// Mitsubishi GX Works2 project: wor01052023   PLC: FX3G

// global labels: Global1
VAR_GLOBAL
  X_3 AT X003 : BOOL;
  Temp_Under15 AT X002 : BOOL;
  Machine_On AT Y004 : BOOL;
  Force_Stop AT X005 : BOOL;
  Cream_Storage AT D1145 : INT;
  M_19 AT M19 : BOOL;
  M_18 AT M18 : BOOL;
END_VAR
VAR_GLOBAL CONSTANT
  biscuits_6 : INT := 6;
END_VAR
VAR_GLOBAL
  biscuits_storage AT D1150 : INT;
  Camera_sensor AT X004 : BOOL;
  Touch_sensor AT X001 : BOOL;
  M_20 AT M20 : BOOL;
  Move_cream AT X011 : BOOL;
  Y_1 AT Y001 : BOOL;
  M_8 AT M8 : BOOL;
END_VAR
VAR_GLOBAL CONSTANT
  RE_timer1 : INT := 10;
END_VAR
VAR_GLOBAL
  TC4_lights AT TC4 : BOOL;
  Y_0 AT Y000 : BOOL;
  TC5_lights AT TC5 : BOOL;
  TS5 AT TS5 : BOOL;
  TC1_lights AT TC1 : BOOL;
  TS1 AT TS1 : BOOL;
END_VAR
VAR_GLOBAL CONSTANT
  RE_timer2 : INT := 40;
END_VAR
VAR_GLOBAL
  M_9 AT M9 : BOOL;
  TS4 AT TS4 : BOOL;
  Chocolate_Container AT D1138 : INT;
  Icing_container AT D1120 : INT;
  Input_chocolate AT D2000 : INT;
  Input_icing AT D2100 : INT;
  Input_biscuits AT D2200 : INT;
  M_88 AT M88 : BOOL;
  Min_chocolate AT D2300 : INT;
  Min_Icing AT D2400 : INT;
  Min_biscuits AT D2500 : INT;
END_VAR
VAR_GLOBAL CONSTANT
  Cream_300 : INT := 300;
END_VAR
VAR_GLOBAL
  M_89 AT M89 : BOOL;
  M_90 AT M90 : BOOL;
  M_91 AT M91 : BOOL;
  CC_0 AT CC0 : BOOL;
  CC_1 AT CC1 : BOOL;
  M_111 AT M111 : BOOL;
  M_112 AT M112 : BOOL;
END_VAR
VAR_GLOBAL CONSTANT
  Double_Cover240 : INT := 240;
  Min_1 : INT := 1;
END_VAR
VAR_GLOBAL
  Y_7 AT Y007 : BOOL;
  Start_day AT X007 : BOOL;
  M_404 AT M404 : BOOL;
  X_10 AT X010 : BOOL;
  X_0 AT X000 : BOOL;
  Counter_5 AT CC5 : BOOL;
END_VAR
VAR_GLOBAL CONSTANT
  RE_counter : INT := 5;
END_VAR
VAR_GLOBAL
  CS5_counter AT CS5 : BOOL;
  Y_2 AT Y002 : BOOL;
  Counter_1 AT CC1 : BOOL;
END_VAR
VAR_GLOBAL CONSTANT
  RE_counter1 : INT := 1;
END_VAR
VAR_GLOBAL
  Counter_6 AT CC6 : BOOL;
END_VAR
VAR_GLOBAL CONSTANT
  RE_count6 : INT := 6;
END_VAR
VAR_GLOBAL
  CS6_downCounter AT CS6 : BOOL;
  finish_packing AT M16 : BOOL;  (* after packing 6 creamBos we will send a signal to add them to the total *)
  analog_output AT D8282 : INT;
  M_17 AT M17 : BOOL;  (* after packing 6 creamBos we will send a signal to add them to the total *)
END_VAR
VAR_GLOBAL CONSTANT
  CreamBo_Unit : INT := 6;
END_VAR
VAR_GLOBAL
  Y_3 AT Y003 : BOOL;
  global_num_CreamBos AT D1234 : INT;
END_VAR
VAR_GLOBAL CONSTANT
  Const_10 : INT := 10;
END_VAR
VAR_GLOBAL
  end_of_day AT M200 : BOOL;
  M_301 AT M301 : BOOL;
  TC11_lights AT TC11 : BOOL;
END_VAR
VAR_GLOBAL CONSTANT
  RE_timer11 : INT := 40;
END_VAR
VAR_GLOBAL
  TS11 AT TS11 : BOOL;
  M_500 AT M500 : BOOL;
  M_501 AT M501 : BOOL;
  TS12 AT TS12 : BOOL;
  TC12_lights AT TC12 : BOOL;
END_VAR
VAR_GLOBAL CONSTANT
  RE_timer12 : INT := 10;
END_VAR
VAR_GLOBAL
  TS13 AT TS13 : BOOL;
  M_505 AT M505 : BOOL;
  TC13_lights AT TC13 : BOOL;
END_VAR
VAR_GLOBAL CONSTANT
  RE_timer13 : INT := 10;
END_VAR
VAR_GLOBAL
  X_6 AT X006 : BOOL;
  Analog_Input AT D8280 : INT;
  TC_DipTimer AT TC20 : BOOL;
END_VAR
VAR_GLOBAL CONSTANT
  RE_5secTimer : INT := 50;  (* 50 mili seconds is 5 seconds *)
END_VAR
VAR_GLOBAL
  TS1_timer AT TS20 : BOOL;
END_VAR
VAR_GLOBAL CONSTANT
  constant6 : INT := 6;
  constant5 : INT := 5;
END_VAR
VAR_GLOBAL
  Container_Dip AT D1139 : INT;
END_VAR
VAR_GLOBAL CONSTANT
  Regular_Cover120 : INT := 120;
END_VAR
VAR_GLOBAL
  M_101 AT M101 : BOOL;
  Y_4 AT Y004 : BOOL;
  M_120 AT M120 : BOOL;
  M_99 AT M99 : BOOL;
  M_113 AT M113 : BOOL;
  M_102 AT M102 : BOOL;
  CS_0 AT CS0 : BOOL;
  CS_1 AT CS1 : BOOL;
  M_300 AT M300 : BOOL;
END_VAR
VAR_GLOBAL CONSTANT
  constant_390 : INT := 390;
END_VAR
VAR_GLOBAL
  Input_moveNew AT D2270 : INT;
  M_75 AT M75 : BOOL;
  TS20_timer AT TS20 : BOOL;
  M_405 AT M405 : BOOL;
  M_321 AT M321 : BOOL;
  M_322 AT M322 : BOOL;
  M_323 AT M323 : BOOL;
  M_324 AT M324 : BOOL;
  M_325 AT M325 : BOOL;
  output_test AT D1237 : INT;
  output_mul AT D1238 : INT;
  M_80 AT M80 : BOOL;
  M_333 AT M333 : BOOL;
END_VAR

// task Task_01 (event TRUE, interval 0, priority 31): POU_01

PROGRAM POU_01
VAR
  M_0 : BOOL;
  TS2 : BOOL;
END_VAR
(* structured ladder/FBD written out as ST: instructions are called as NAME(EN, inputs, outputs); _pN, _eN, _tN stand for wires *)
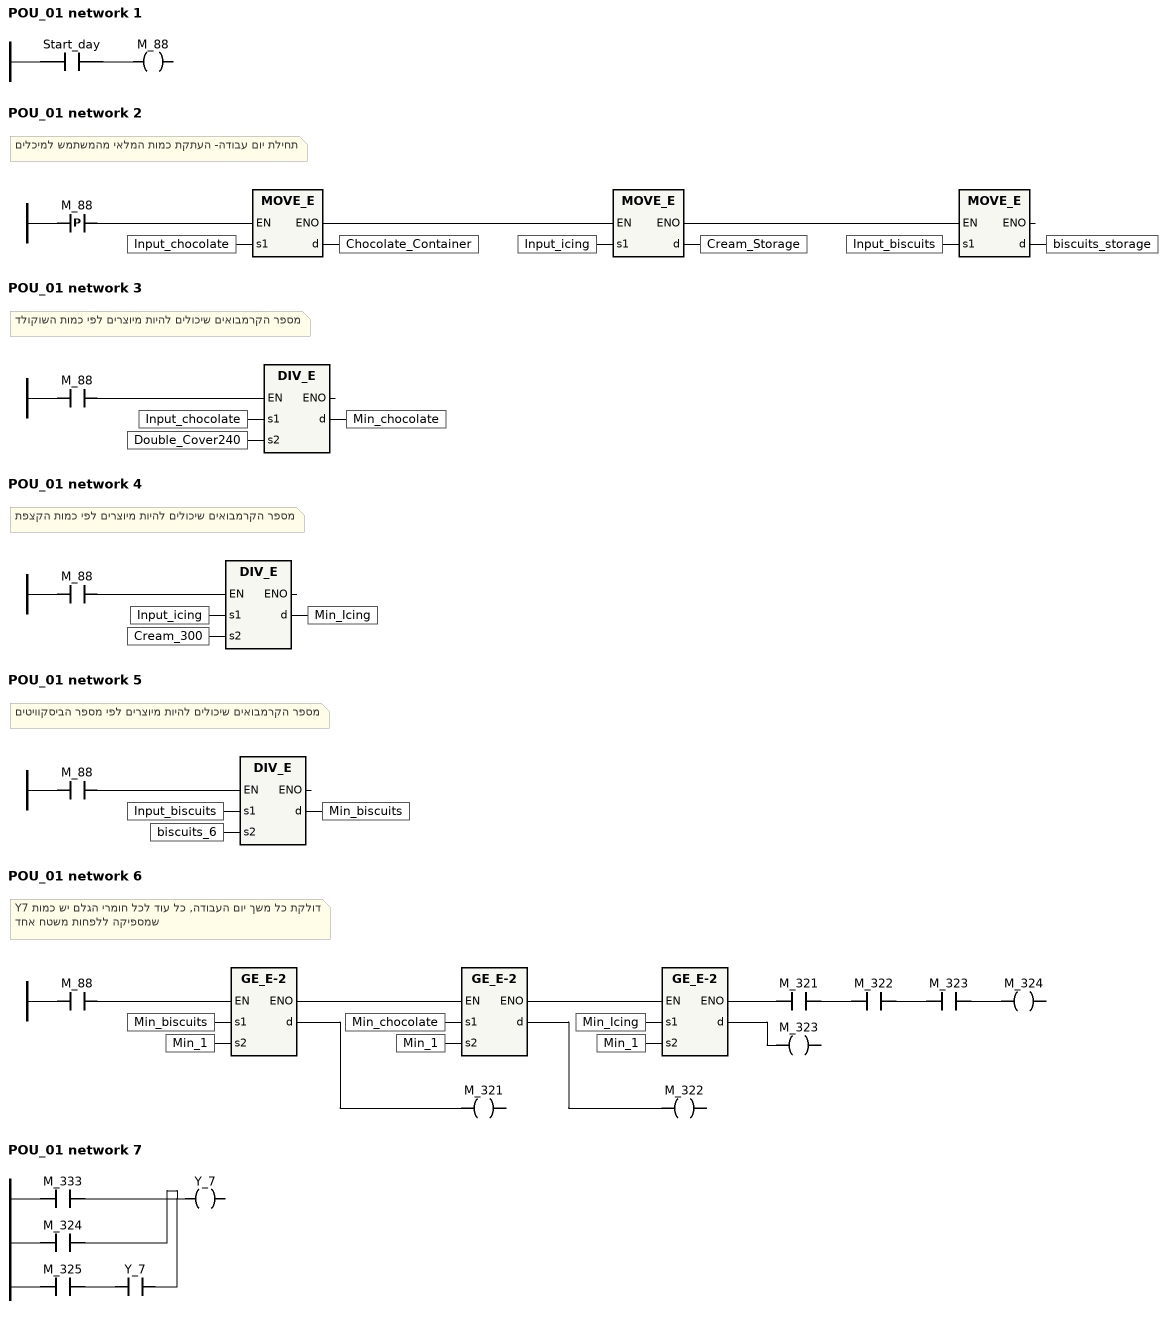
(* network 1 *)
M_88 := Start_day;
(* network 2 *)
(* תחילת יום עבודה- העתקת כמות המלאי מהמשתמש למיכלים *)
_e1 := MOVE_E(LDP(TRUE, M_88), Input_chocolate, Chocolate_Container);
_e2 := MOVE_E(_e1, Input_icing, Cream_Storage);
MOVE_E(_e2, Input_biscuits, biscuits_storage);
(* network 3 *)
(* מספר הקרמבואים שיכולים להיות מיוצרים לפי כמות השוקולד *)
DIV_E(M_88, Input_chocolate, Double_Cover240, Min_chocolate);
(* network 4 *)
(* מספר הקרמבואים שיכולים להיות מיוצרים לפי כמות הקצפת *)
DIV_E(M_88, Input_icing, Cream_300, Min_Icing);
(* network 5 *)
(* מספר הקרמבואים שיכולים להיות מיוצרים לפי מספר הביסקוויטים *)
DIV_E(M_88, Input_biscuits, biscuits_6, Min_biscuits);
(* network 6 *)
(* Y7 דולקת כל משך יום העבודה, כל עוד לכל חומרי הגלם יש כמות שמספיקה ללפחות משטח אחד *)
_e2 := GE_E(M_88, Min_biscuits, Min_1, _t1);
_e4 := GE_E(_e2, Min_chocolate, Min_1, _t3);
_e6 := GE_E(_e4, Min_Icing, Min_1, _t5);
M_324 := _e6 AND M_321 AND M_322 AND M_323;
M_321 := _t1;
M_323 := _t5;
M_322 := _t3;
(* network 7 *)
Y_7 := M_333 OR M_324 OR (M_325 AND Y_7);
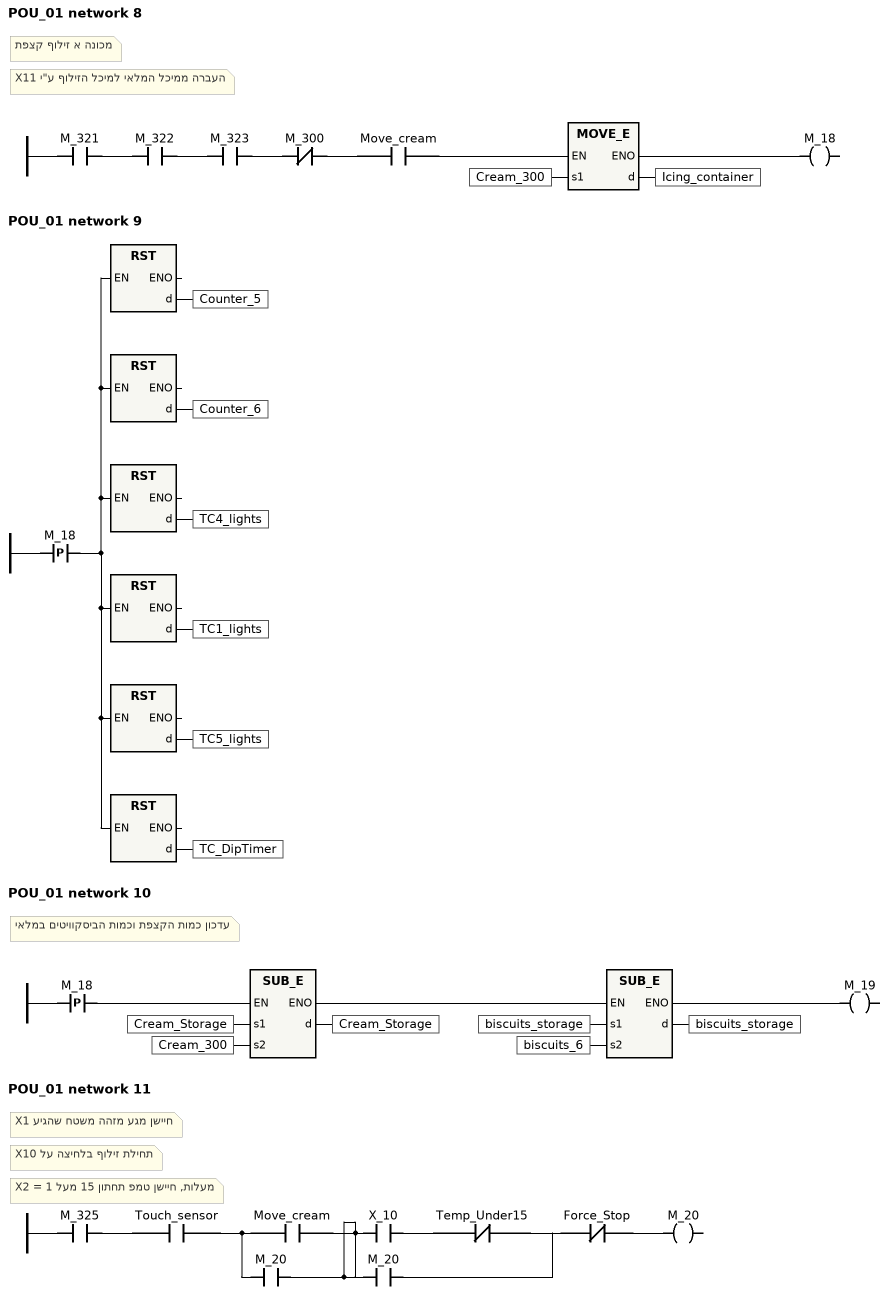
(* network 8 *)
(* מכונה א זילוף קצפת *)
(* העברה ממיכל המלאי למיכל הזילוף ע"י X11 *)
_e1 := MOVE_E(M_321 AND M_322 AND M_323 AND NOT M_300 AND Move_cream, Cream_300, Icing_container);
M_18 := _e1;
(* network 9 *)
_p1 := LDP(TRUE, M_18);
RST(_p1, Counter_5);
RST(_p1, Counter_6);
RST(_p1, TC4_lights);
RST(_p1, TC1_lights);
RST(_p1, TC5_lights);
RST(_p1, TC_DipTimer);
(* network 10 *)
(* עדכון כמות הקצפת וכמות הביסקוויטים במלאי *)
_e1 := SUB_E(LDP(TRUE, M_18), Cream_Storage, Cream_300, Cream_Storage);
_e2 := SUB_E(_e1, biscuits_storage, biscuits_6, biscuits_storage);
M_19 := _e2;
(* network 11 *)
(* חיישן מגע מזהה משטח שהגיע X1 *)
(* תחילת זילוף בלחיצה על X10 *)
(* X2 = 1 מעל 15 מעלות, חיישן טמפ תחתון *)
_p1 := M_325 AND Touch_sensor;
_p2 := (_p1 AND Move_cream) OR (_p1 AND M_20);
M_20 := ((_p2 AND X_10 AND NOT Temp_Under15) OR (_p2 AND M_20)) AND NOT Force_Stop;
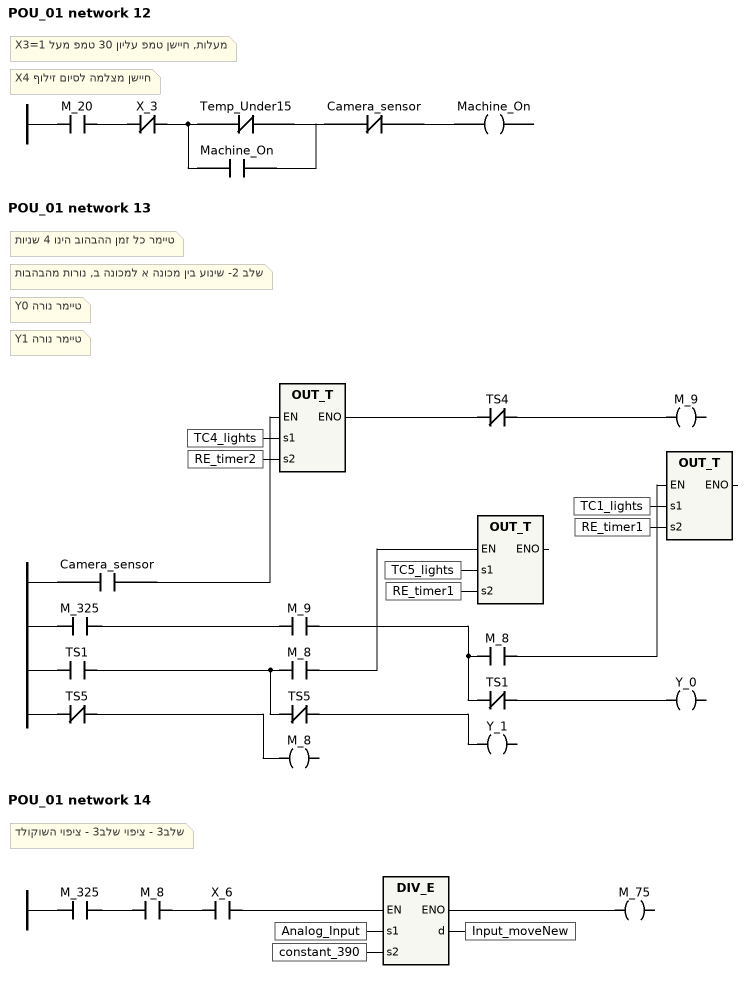
(* network 12 *)
(* X3=1 טמפ מעל 30 מעלות, חיישן טמפ עליון *)
(* חיישן מצלמה לסיום זילוף X4 *)
_p1 := M_20 AND NOT X_3;
Machine_On := ((_p1 AND NOT Temp_Under15) OR (_p1 AND Machine_On)) AND NOT Camera_sensor;
(* network 13 *)
(* טיימר כל זמן ההבהוב הינו 4 שניות *)
(* שלב 2- שינוע בין מכונה א למכונה ב, נורות מהבהבות *)
(* טיימר נורה Y0 *)
(* טיימר נורה Y1 *)
_e1 := OUT_T(Camera_sensor, TC4_lights, RE_timer2);
M_9 := _e1 AND NOT TS4;
_p2 := M_325 AND M_9;
OUT_T(_p2 AND M_8, TC1_lights, RE_timer1);
Y_0 := _p2 AND NOT TS1;
OUT_T(TS1 AND M_8, TC5_lights, RE_timer1);
Y_1 := TS1 AND NOT TS5;
M_8 := NOT TS5;
(* network 14 *)
(* שלב3 - ציפוי שלב3 - ציפוי השוקולד *)
_e1 := DIV_E(M_325 AND M_8 AND X_6, Analog_Input, constant_390, Input_moveNew);
M_75 := _e1;
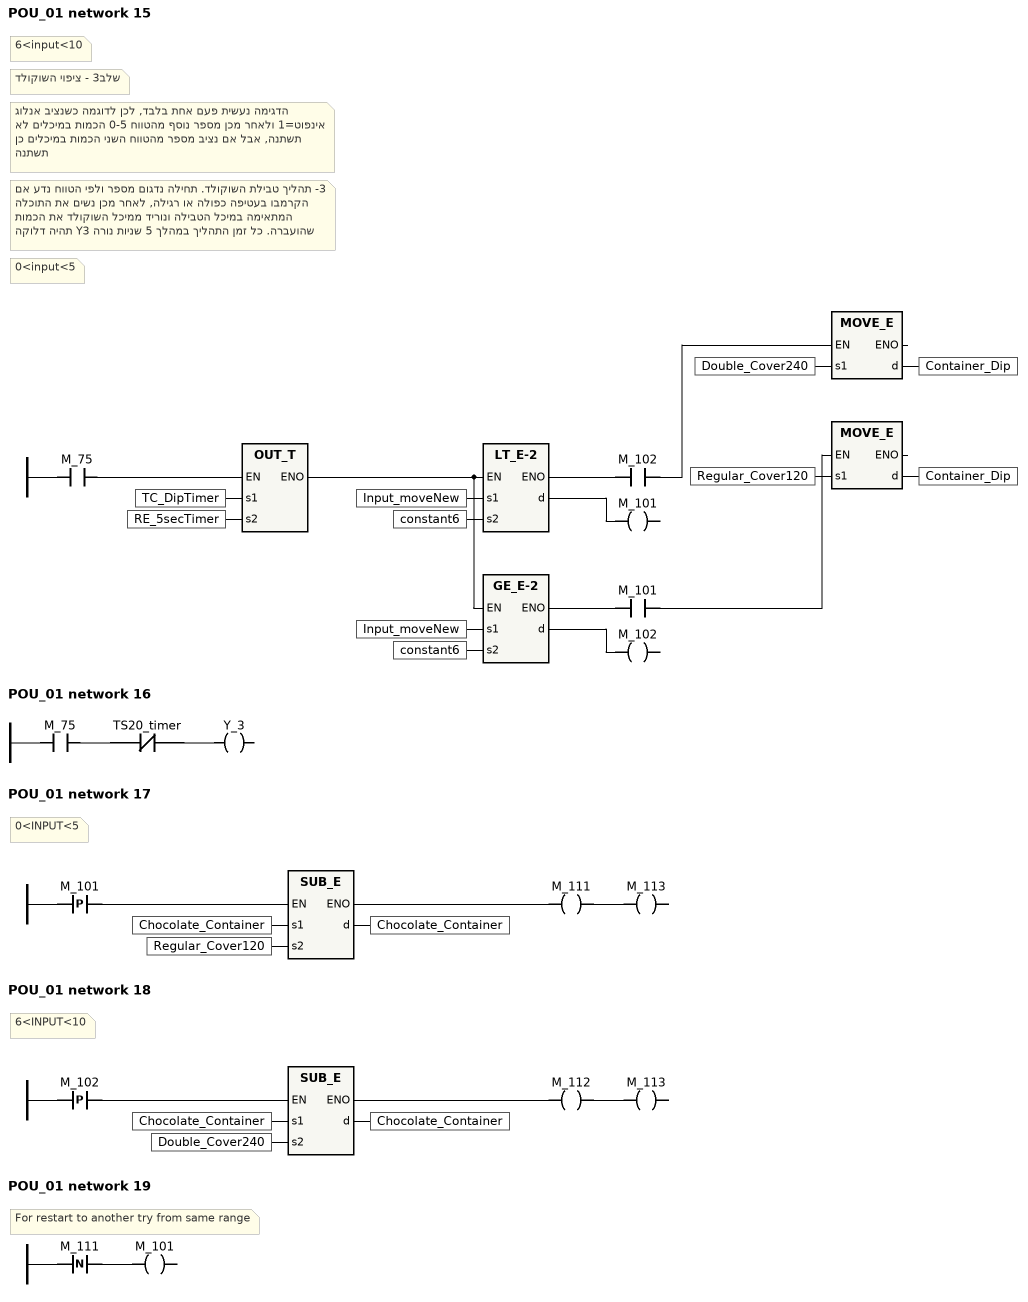
(* network 15 *)
(* 6<input<10 *)
(* שלב3 - ציפוי השוקולד *)
(* הדגימה נעשית פעם אחת בלבד, לכן לדוגמה כשנציב אנלוג אינפוט=1 ולאחר מכן מספר נוסף מהטווח 0-5 הכמות במיכלים לא תשתנה, אבל אם נציב מספר מהטווח השני הכמות במיכלים כן תשתנה *)
(* 3- תהליך טבילת השוקולד. תחילה נדגום מספר ולפי הטווח נדע אם הקרמבו בעטיפה כפולה או רגילה, לאחר מכן נשים את התוכלה המתאימה במיכל הטבילה ונוריד ממיכל השוקולד את הכמות שהועברה. כל זמן התהליך במהלך 5 שניות נורה Y3 תהיה דלוקה *)
(* 0<input<5 *)
_e1 := OUT_T(M_75, TC_DipTimer, RE_5secTimer);
_e3 := LT_E(_e1, Input_moveNew, constant6, _t2);
MOVE_E(_e3 AND M_102, Double_Cover240, Container_Dip);
M_101 := _t2;
_e5 := GE_E(_e1, Input_moveNew, constant6, _t4);
MOVE_E(_e5 AND M_101, Regular_Cover120, Container_Dip);
M_102 := _t4;
(* network 16 *)
Y_3 := M_75 AND NOT TS20_timer;
(* network 17 *)
(* 0<INPUT<5 *)
_e1 := SUB_E(LDP(TRUE, M_101), Chocolate_Container, Regular_Cover120, Chocolate_Container);
M_111 := _e1;
M_113 := _e1;
(* network 18 *)
(* 6<INPUT<10 *)
_e1 := SUB_E(LDP(TRUE, M_102), Chocolate_Container, Double_Cover240, Chocolate_Container);
M_112 := _e1;
M_113 := _e1;
(* network 19 *)
(* For restart to another try from same range *)
M_101 := LDF(TRUE, M_111);
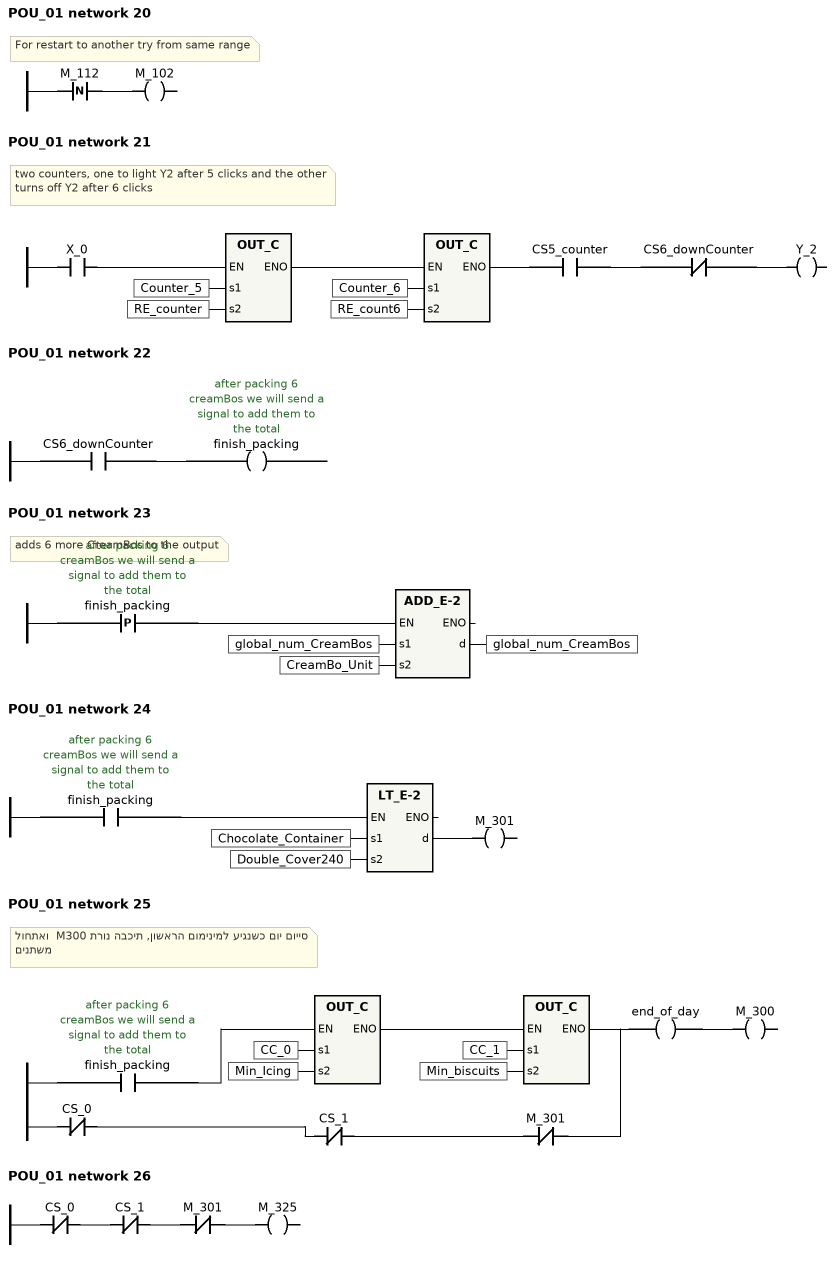
(* network 20 *)
(* For restart to another try from same range *)
M_102 := LDF(TRUE, M_112);
(* network 21 *)
(* two counters, one to light Y2 after 5 clicks and the other turns off Y2 after 6 clicks *)
_e1 := OUT_C(X_0, Counter_5, RE_counter);
_e2 := OUT_C(_e1, Counter_6, RE_count6);
Y_2 := _e2 AND CS5_counter AND NOT CS6_downCounter;
(* network 22 *)
finish_packing := CS6_downCounter;
(* network 23 *)
(* adds 6 more CreamBos to the output *)
ADD_E(LDP(TRUE, finish_packing), global_num_CreamBos, CreamBo_Unit, global_num_CreamBos);
(* network 24 *)
LT_E(finish_packing, Chocolate_Container, Double_Cover240, _t1);
M_301 := _t1;
(* network 25 *)
(* סייום יום כשנגיע למינימום הראשון, תיכבה נורת M300  ואתחול משתנים *)
_e1 := OUT_C(finish_packing, CC_0, Min_Icing);
_e2 := OUT_C(_e1, CC_1, Min_biscuits);
_p3 := _e2 OR (NOT CS_0 AND NOT CS_1 AND NOT M_301);
end_of_day := _p3;
M_300 := _p3;
(* network 26 *)
M_325 := NOT CS_0 AND NOT CS_1 AND NOT M_301;
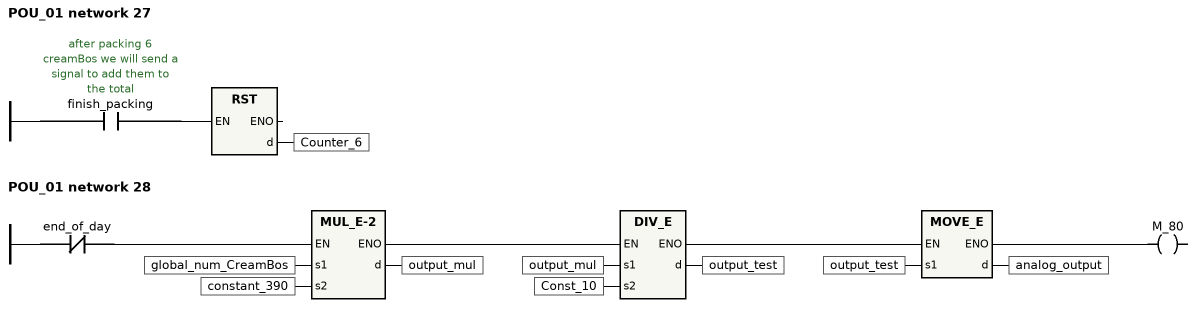
(* network 27 *)
RST(finish_packing, Counter_6);
(* network 28 *)
_e1 := MUL_E(NOT end_of_day, global_num_CreamBos, constant_390, output_mul);
_e2 := DIV_E(_e1, output_mul, Const_10, output_test);
_e3 := MOVE_E(_e2, output_test, analog_output);
M_80 := _e3;
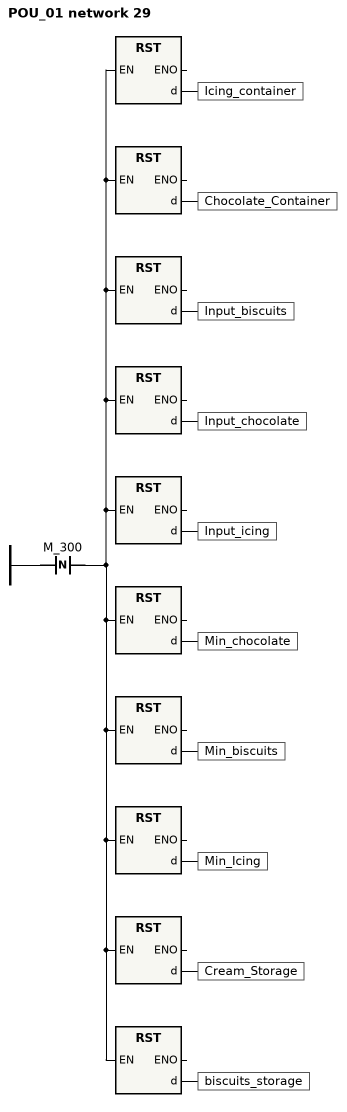
(* network 29 *)
_p1 := LDF(TRUE, M_300);
RST(_p1, Icing_container);
RST(_p1, Chocolate_Container);
RST(_p1, Input_biscuits);
RST(_p1, Input_chocolate);
RST(_p1, Input_icing);
RST(_p1, Min_chocolate);
RST(_p1, Min_biscuits);
RST(_p1, Min_Icing);
RST(_p1, Cream_Storage);
RST(_p1, biscuits_storage);
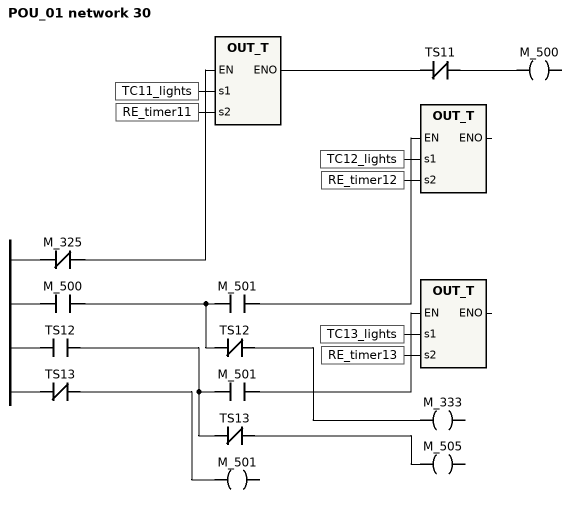
(* network 30 *)
_e1 := OUT_T(NOT M_325, TC11_lights, RE_timer11);
M_500 := _e1 AND NOT TS11;
OUT_T(M_500 AND M_501, TC12_lights, RE_timer12);
M_333 := M_500 AND NOT TS12;
OUT_T(TS12 AND M_501, TC13_lights, RE_timer13);
M_505 := TS12 AND NOT TS13;
M_501 := NOT TS13;
END_PROGRAM
